// TIA Portal V18 export
FUNCTION_BLOCK "SlewInc"   // FB122, LAD
TITLE = SlewInc
{ S7_Optimized_Access := 'TRUE' }
// Written BY Kristopher Gimenez Feb 17,2023
// This block will be used to slew the output but the at the set rate per second base on input slew rate
// stored: AutoNumber false, MemoryReserve 100, SetENOAutomatically false
   VAR_INPUT
      SlewRate : Real;   // Slew rate in mA/sec
   END_VAR
   VAR_IN_OUT
      RealValue : Real;
   END_VAR
   VAR
      Slew : Bool;
      Inc_TON : TON_TIME;
   END_VAR
   VAR_TEMP
      tempReal : Real;
   END_VAR
BEGIN

REGION Network 1: Slew rate in mA/sec
   // Increase the input value by the slew rate
   // Increasing every 10ms divide rate by 100
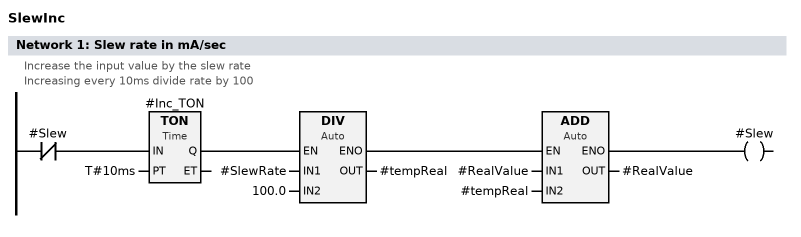
   RUNG wire#powerrail
      I_Contact( #Slew )
      { S7_Templates := "time_type := Time" } #Inc_TON.TON(pt := T#10ms, et =>)
      Div(in1 := #SlewRate, in2 := 100.0, out => #tempReal)
      Add(in1 := #RealValue, in2 := #tempReal, out => #RealValue)
      Coil( #Slew )
   END_RUNG
   // the same network as SCL:
   #Inc_TON(IN := NOT #Slew, PT := T#10ms);   // TON
   IF #Inc_TON.Q THEN
       #tempReal := #SlewRate / 100.0;
       #RealValue := #RealValue + #tempReal;
   END_IF;
   #Slew := #Inc_TON.Q;
END_REGION
END_FUNCTION_BLOCK
